Fanuc KAREL source: kt00904.KL

PROGRAM KT00904
%STACKSIZE=65535
%PRIORITY=65535
%NOLOCKGROUP
VAR
P1 : XYZWPR
P2 : XYZWPR
-- UNRESOLVED DECLARATIONS (source type spelling not recovered)
-- OUT : TYPE_0x0013 (type_u16=0x0013)
BEGIN
P1.X=1.0
P2.Y=2.0
P1.X=1.0
P2.Y=2.0
-- UNSAFE_SOURCE_IR line 13: OUT = APPROACH(convert_xyzwpr_to_position(P1))
END KT00904
